// TIA Portal V16 export
// export: Created 2021-07-12T14:47:19.2973696Z, ExportSetting WithDefaults, DisplayName Totally Integrated Automation Portal, DisplayVersion V16, DisplayName TIA Portal Version Control Interface, DisplayVersion V16, DisplayName TIA Portal Openness, DisplayVersion V16, DisplayName STEP 7 Professional, DisplayVersion V16, DisplayName STEP 7 Safety, DisplayVersion V16, DisplayName WinCC Professional, DisplayVersion V16
TYPE "LSimaHydTO_typeStatusServo"
TITLE = LSimaHydTO_typeStatusServo
// Indicates the status of position control
// stored: IsFailsafeCompliant false
   STRUCT
      BalancedPosition { ExternalWritable := 'False'} : LReal;   // Position after the balancing filter
      ControlDifference { ExternalWritable := 'False'} : LReal;   // Control error
   END_STRUCT;
END_TYPE
